com_read(com:= m26_handle, rbuffer := ADR(lac_read_buffer), rsize := SIZEOF(lac_read_buffer));

END_FUNCTION_BLOCK

// MIC7001/Application/j1939/PGN_F004_RPM
FUNCTION_BLOCK PGN_F004_RPM
VAR_INPUT
	ID,mask:DWORD;
	TData    : ARRAY[0..7] OF BYTE; 
	new_data : BOOL := FALSE;
END_VAR
VAR_OUTPUT
	RPM: UINT;
	torque:UINT;
END_VAR
VAR
	Timeout: TON:=(IN:=TRUE , PT:=T#200ms );
	temp_rpm:UINT;
END_VAR


Timeout();
IF Timeout.Q THEN;
	RPM := 0;
	torque := 0;
END_IF

IF new_data THEN
	Timeout(IN:=FALSE );
	Timeout.IN:=TRUE;
ELSE
	RETURN;
END_IF

IF((ID AND MASK) = 16#00F00400) THEN
	rpm := (TData[3] + TData[4]*256)/8;
	torque := TData[2] - 125;
END_IF

END_FUNCTION_BLOCK

// MIC7001/Application/j1939/PGN_FEEE_TEMP
FUNCTION_BLOCK PGN_FEEE_TEMP
VAR_INPUT
	ID,mask:DWORD;
	TData    : ARRAY[0..7] OF BYTE; 
	new_data : BOOL := FALSE;
END_VAR
VAR_OUTPUT
	Eng_Coolaant_Temp:INT;(*spn 110*)
	Eng_Fuel_Temp:INT;(*spn 174*)
	Eng_Oil_Temp:INT;(*spn 175*)
	Turbo_Oil_Temp:INT;(*spn 176*)
	Eng_InterCooler_Temp:INT;(*spn 52*)
	Eng_InterCooler_Thermostat_Opening:BYTE;(*spn 1134*)
	MeasNotValid:BYTE;
	Error: BYTE;
END_VAR
VAR
	Timeout: TON:=(IN:=TRUE , PT:=T#2s );
END_VAR

Timeout();
IF((ID AND MASK) = 16#00FEEE00) THEN
	Eng_Coolaant_Temp:=temp_neg40_to_210oC(TData[0]);
	Eng_Fuel_Temp:=temp_neg40_to_210oC(TData[1]);
	Eng_Oil_Temp:=temp_absZero_to_1735oC(TData[2]+TData[3]*16#100);
	Turbo_Oil_Temp:=temp_absZero_to_1735oC(TData[4]+TData[5]*16#100);
	Eng_InterCooler_Temp:=temp_neg40_to_210oC(TData[6]);
	Eng_InterCooler_Thermostat_Opening:=pros100(TData[7]);
	MeasNotValid:=PACK(TData[0]>16#FA, TData[1]>16#FA, TData[3]>16#FA, TData[5]>16#FA, TData[6]>16#FA, TData[7]>16#FA, FALSE, FALSE);

	Error:=PACK(TData[0]=16#FE, TData[1]=16#FE, TData[3]=16#FE, TData[5]=16#FE, TData[6]=16#FE, TData[7]=16#FE, FALSE, FALSE);
	IF new_data THEN
		Timeout(IN:=FALSE );
		Timeout.IN:=TRUE;
	END_IF

END_IF

IF Timeout.Q THEN;
	Eng_Coolaant_Temp:=0;
	Eng_Fuel_Temp:=0;
	Eng_Oil_Temp:=0;
	Turbo_Oil_Temp:=0;
	Eng_InterCooler_Temp:=0;
	Eng_InterCooler_Thermostat_Opening:=0;
END_IF

END_FUNCTION_BLOCK

// MIC7001/Application/j1939/PACK
FUNCTION PACK : BYTE
VAR_INPUT
	bit0:BOOL;
	bit1:BOOL;
	bit2:BOOL;
	bit3:BOOL;
	bit4:BOOL;
	bit5:BOOL;
	bit6:BOOL;
	bit7:BOOL;
END_VAR
VAR
END_VAR

PACK := 0;
IF bit0 THEN
	PACK := PACK + 1;
END_IF

IF bit1 THEN
	PACK := PACK + 2;
END_IF

IF bit2 THEN
	PACK := PACK + 4;
END_IF

IF bit3 THEN
	PACK := PACK + 8;
END_IF

IF bit4 THEN
	PACK := PACK + 16;
END_IF

IF bit5 THEN
	PACK := PACK + 32;
END_IF

IF bit6 THEN
	PACK := PACK + 64;
END_IF

IF bit7 THEN
	PACK := PACK + 128;
END_IF

END_FUNCTION

// MIC7001/Application/functions/fn_get_Q_221ma
FUNCTION fn_get_Q_221ma : real
VAR_INPUT
	press:REAL;
END_VAR
VAR
	q:REAL;
END_VAR

IF press < 5.1 THEN
	q := 126.0;
ELSIF press < 14.1 THEN
	q := 126.0 + (press-5.1)*(71.0-126.0)/(14.1-5.1);
ELSIF press < 34.3 THEN
	q := 71.0 + (press-14.1)*(35.0-71.0)/(34.3-14.1);
ELSE
	q := 35.0;
END_IF

fn_get_Q_221ma := q;

END_FUNCTION

// MIC7001/Application/functions/fn_get_Q_408ma
FUNCTION fn_get_Q_408ma : real
VAR_INPUT
	press:REAL;
END_VAR
VAR
	q:REAL;
END_VAR

IF press < 11.4 THEN
	q := 125.0;
ELSIF press < 20.3 THEN
	q := 125.0 + (press-11.4)*(69.0-125.0)/(20.3-11.4);
ELSIF press < 34.3 THEN
	q := 69.0 + (press-20.3)*(35.0-69.0)/(34.3-20.3);
ELSE
	q := 35.0;
END_IF

fn_get_Q_408ma := q;

END_FUNCTION

// MIC7001/Application/functions/fn_get_Q_631ma
FUNCTION fn_get_Q_631ma : real
VAR_INPUT
	press:REAL;
END_VAR
VAR
	q:REAL;
END_VAR

IF press < 21.1 THEN
	q := 124.0;
ELSIF press < 30.0 THEN
	q := 124.0 + (press-21.1)*(67.0-124.0)/(30.0-21.1);
ELSIF press < 34.3 THEN
	q := 67.0 + (press-30.0)*(57.0-67.0)/(34.3-30.0);
ELSE
	q := 57.0;
END_IF

fn_get_Q_631ma := q;

END_FUNCTION

// MIC7001/Application/functions/fn_get_Q_521ma
FUNCTION fn_get_Q_521ma : real
VAR_INPUT
	press:REAL;
END_VAR
VAR
	q:REAL;
END_VAR

IF press < 16.2 THEN
	q := 125.0;
ELSIF press < 25.2 THEN
	q := 125.0 + (press-16.2)*(68.0-125.0)/(25.2-16.2);
ELSIF press < 34.3 THEN
	q := 68.0 + (press-25.2)*(46.0-68.0)/(34.3-25.2);
ELSE
	q := 46.0;
END_IF

fn_get_Q_521ma := q;

END_FUNCTION

// MIC7001/Application/parameters/FB_PARA_REAL
FUNCTION_BLOCK FB_PARA_REAL
VAR_INPUT
	enable:BOOL := FALSE;
	clear:BOOL := FALSE;
	pPara:POINTER TO DUT_PARA_REAL;
END_VAR

VAR_OUTPUT
	ok:BOOL := FALSE;
	zero:BOOL := FALSE;
END_VAR

VAR
	hFile: RTS_IEC_HANDLE := 0;
	sync:BOOL := FALSE;  
	stat:UINT:= 0;
	
	i :UINT;
	str:STRING(1024);
END_VAR


IF NOT enable OR pPara^.num < 1 THEN
	stat := 0;
	RETURN;
END_IF

CASE stat OF
	0:  //init
		IF rd_all(pPara^.filename)	THEN 
			zero := FALSE;
			stat := 10;
		ELSE
			clear_all();
			IF wr_all(pPara^.filename) THEN
				zero := TRUE;
				stat := 10;
			END_IF
		END_IF
	
	10: // normal
		IF chk_chg() THEN
			ok := FALSE;
			IF wr_all(pPara^.filename) THEN
				ok := TRUE;
				zero := FALSE;
			END_IF
		END_IF	
		
		IF clear THEN
			clear_all();
			IF wr_all(pPara^.filename) THEN
				zero := TRUE;
			END_IF
		END_IF
END_CASE

METHOD rd_all : bool
VAR_INPUT
	filename:STRING(256);
END_VAR

VAR
	iNumber:INT;
	udiByteRead:LWORD;
	udiPos:UDINT;
	udiOpenError: RTS_IEC_RESULT;
	udiReadError: RTS_IEC_RESULT;
	str: STRING(255);
	ulOffset:DWORD;
	batch: BOOL;
	check_sum :REAL;
END_VAR
rd_all := FALSE;

hFile := sysfileopen(szFile := filename, am := sysfile.AM_READ, pResult:= ADR(udiOpenError));
IF hFile = RTS_INVALID_HANDLE THEN
	RETURN;
END_IF

ulOffset := 0;
batch := TRUE;

check_sum := 0.0;
FOR i := 1 TO pPara^.num DO
	IF udiByteRead < 50 AND batch THEN
		udiPos := SysFileSetPos(hFile:=hFile, ulOffset := ulOffset);
		udiByteRead := sysfile.SysFileRead(hfile := hFile,pbyBuffer := ADR(str), ulSize := 255 , pResult := ADR(udiReadError));
		IF udiByteRead < 255 THEN
			batch := FALSE;
		END_IF
	END_IF
	IF udiByteRead < 1 THEN  //读取失败
		sysfile.SysFileClose(hFile := hFile);
		RETURN;
	END_IF

	iNumber := find(str, '$N');
	IF iNumber < 2 THEN
		sysfile.SysFileClose(hFile := hFile);
		RETURN;
	END_IF
	
	pPara^.para[i] := STRING_TO_REAL(left(str,iNumber-1));
	str := delete(str, iNumber,1);
	pPara^.old_val[i] := pPara^.para[i];
	
	udiByteRead := udiByteRead - ANY_TO_LWORD(iNumber);
	ulOffset := ulOffset + ANY_TO_DWORD(iNumber);

	IF i = pPara^.num THEN
		IF ABS(check_sum-pPara^.para[i]) > 0.01 THEN
			RETURN;  //error
		END_IF
	ELSE
		check_sum := check_sum + pPara^.para[i];
	END_IF
END_FOR

sysfile.SysFileClose(hFile := hFile);
rd_all := TRUE;
END_METHOD

METHOD chk_chg : bool
VAR_INPUT
END_VAR

VAR
	i :UINT;
END_VAR
chk_chg := TRUE;

FOR i := 1 TO pPara^.num  DO
	IF pPara^.para[i] <> pPara^.old_val[i] THEN
		RETURN;
	END_IF
END_FOR

chk_chg := FALSE;
END_METHOD

METHOD clear_all : bool
VAR_INPUT
	
END_VAR
FOR i := 1 TO pPara^.num DO
	pPara^.para[i] := 0.0;
	pPara^.old_val[i] := 0.0;
END_FOR

clear_all := TRUE;
END_METHOD

METHOD wr_all : bool
VAR_INPUT
	filename:STRING(256);
END_VAR

VAR
	iNumber:INT;
	udiByteWrite:LWORD;
	udiPos:UDINT;
	udiOpenError: RTS_IEC_RESULT;
	udiWriteError: RTS_IEC_RESULT;
	str_size:DWORD;
	check_sum: REAL;
END_VAR
wr_all := FALSE;
hFile := sysfileopen(szFile := filename, am := sysfile.AM_WRITE, pResult := ADR(udiOpenError));
IF hFile = RTS_INVALID_HANDLE THEN
	RETURN;
END_IF

udiPos := SysFileSetPos(hFile:=hFile, ulOffset := 0);

check_sum := 0.0;
str:= ANY_TO_STRING('');
FOR i := 1 TO pPara^.num DO
	IF i = pPara^.num THEN  //the last val, check_sum
		pPara^.para[i] := check_sum;
	ELSE
		check_sum := check_sum + pPara^.para[i];
	END_IF	
	str := concat(str, ANY_TO_STRING(pPara^.para[i]));
	str := concat(str, ANY_TO_STRING('$N'));
	str_size := ANY_TO_DWORD(len(str));
	IF str_size > 200 THEN
		udiByteWrite := sysfile.SysFileWrite(hFile := hFile,pbyBuffer := ADR(str),ulSize := str_size, pResult := ADR(udiWriteError));
		IF udiByteWrite = str_size THEN
			str := '';
		END_IF
	END_IF	
END_FOR
udiByteWrite := sysfile.SysFileWrite(hFile := hFile,pbyBuffer := ADR(str),ulSize := str_size, pResult := ADR(udiWriteError));
	
IF udiByteWrite <> str_size THEN
	sysfile.SysFileClose(hFile);
	RETURN;
END_IF
sysfile.SysFileClose(hFile);

	
FOR i := 1 TO pPara^.num DO
	pPara^.old_val[i] := pPara^.para[i];
END_FOR

hFile := 0;

wr_all := TRUE;
END_METHOD

END_FUNCTION_BLOCK

// MIC7001/Application/functions/fn_get_mins
FUNCTION fn_get_mins : DWORD
VAR_INPUT
	
END_VAR
VAR
	hFile: RTS_IEC_HANDLE;
	udiOpenError: RTS_IEC_RESULT;
	udiPos: UDINT;
	udiByteRead: __XWORD;
	str: STRING(255);
	udiReadError: RTS_IEC_RESULT;
	i: INT;
	number: INT;
	len_of_number: INT;
	mode: UINT;
	pInMode: INT;
	mins: DWORD;
END_VAR

fn_get_mins := 0;

//检测文件是否存在
hFile := sysfileopen(szFile := gvl.mins_file, am := sysfile.AM_READ, pResult:= ADR(udiOpenError));
IF hFile = RTS_INVALID_HANDLE	THEN  //文件不存在
	RETURN;
END_IF

//文件存在，开始读取内容
udiPos := SysFileSetPos(hFile:=hFile, ulOffset := 0);
udiByteRead := sysfile.SysFileRead(hfile := hFile,pbyBuffer := ADR(str), ulSize := SIZEOF(str), pResult := ADR(udiReadError));
IF udiByteRead < 1 THEN  //读取失败
	sysfile.SysFileClose(hFile := hFile);
	RETURN;
END_IF
sysfile.SysFileClose(hFile);

//读取本行的数字

mins := STRING_TO_DWORD(str);


fn_get_mins := mins;
RETURN;

END_FUNCTION

// MIC7001/Application/Visualization
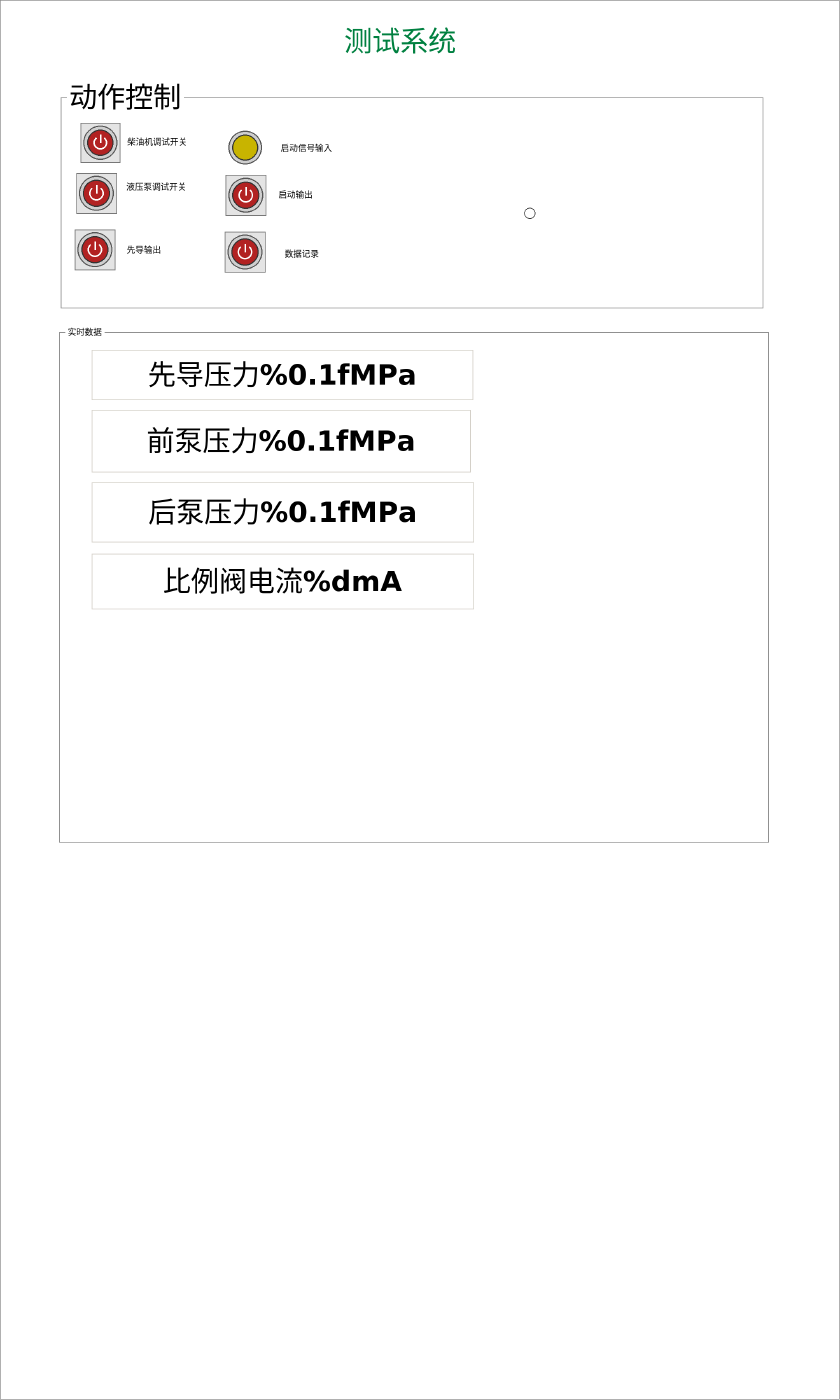
VISUALIZATION Visualization  // 1080x1800
    Label (307,19 415x68), "测试系统"
    GroupBox (78,117 903x279), "动作控制"
        Line (40,109)
        PowerSwitch (20,103 52x57), variable: GVL.g_pump_work, behaviour: TOGGLE, style: Switch-PowerSwitch-Red
        PowerSwitch (23,41 56x51), variable: GVL.g_engine_work, behaviour: TOGGLE, style: Switch-PowerSwitch-Red
        Label (69,47 110x37), "柴油机调试开关"
        Label (68,105 110x37), "液压泵调试开关"
        PowerSwitch (18,177 52x54), variable: GVL.g_do_pilot, behaviour: TOGGLE, style: Switch-PowerSwitch-Red
        Label (72,186 70x37), "先导输出"
        RadioButton (594,47 293x220), variable: g_mode
        PowerSwitch (211,180 52x54), variable: prg_data.data_save, behaviour: TOGGLE, style: Switch-PowerSwitch-Red
        Label (275,191 70x37), "数据记录"
        Lamp1 (212,46 50x53), variable: GVL.DI_start, style: Lamp-Lamp1-Yellow
        Label (270,55 92x37), "启动信号输入"
        PowerSwitch (212,107 52x54), variable: GVL.g_do_start, behaviour: TOGGLE, style: Switch-PowerSwitch-Red
        Label (267,115 70x37), "启动输出"
    GroupBox (76,419 912x664), "实时数据"
        Textfield (42,31 490x64), "先导压力%0.1fMPa", text variable: GVL.g_ai_pilot
        Textfield (42,108 487x80), "前泵压力%0.1fMPa", text variable: GVL.g_ai_press_pump1
        Textfield (42,201 491x77), "后泵压力%0.1fMPa", text variable: GVL.g_ai_press_pump2
        Textfield (42,293 491x71), "比例阀电流%dmA", text variable: GVL.g_ai_curr_prop
END_VISUALIZATION
